FUNCTION_BLOCK FB_AcceleratorLinks
VAR_INPUT

END_VAR

VAR_OUTPUT
END_VAR


VAR

    {attribute 'pytmc' := '
        pv: eEnrg:Hgvpu
        link: BEND:DMPH:400:BACT
        field: EGU GeV
        field: PREC 3
    '}
    fbHgvpuElectronEnergy : FB_LREALFromEPICS;

    {attribute 'pytmc' := '
        pv: eEnrg:SXU
        link: BEND:DMPS:400:BACT
        field: EGU GeV
        field: PREC 3
    '}
    fbSxuElectronEnergy : FB_LREALFromEPICS;

END_VAR

fbHgvpuElectronEnergy();
fbSxuElectronEnergy();

END_FUNCTION_BLOCK

(* stored: Version 1.1.0.1, ProductVersion 3.1.4022.18
   POU FB_AcceleratorLinks: Id {a8c08e7c-c206-478b-9402-da1b879edfc5}, SpecialFunc None *)
